// Feedback belongs to the plant, not to the commanded direction.
TYPE ST_CylinderFeedback :
STRUCT
    advanced : BOOL;
    retracted : BOOL;
END_STRUCT
END_TYPE

(* stored: Version 1.1.0.1
   DUT ST_CylinderFeedback: Id {91abd59d-11ba-4c35-a25a-3cd008fa786e} *)
